// TwinCAT 3 PLC project PLC
// ProgramVersion: 3.1.4024.0
// libraries:
//   Tc2_Standard, * (Beckhoff Automation GmbH)
//   Tc2_System, * (Beckhoff Automation GmbH)
//   Tc3_Module, * (Beckhoff Automation GmbH)
// project tree:
//   / PlcTask.TcTTO
//   POUs/ MAIN.TcPOU
//   POUs/TEMPLATE ST FB%27s/ AdvancedFaultDetection.TcPOU (not stored), Auto_Manual_CycleControl.TcPOU (not stored), CYL.TcPOU (not stored), FB_analog.TcPOU (not stored), FB_Conveyor.TcPOU (not stored), FB_Fan.TcPOU (not stored), FB_FaultDetection.TcPOU (not stored), FB_FlowMeter.TcPOU (not stored), FB_IO_Card_ARRAY.TcPOU (not stored), FB_IO_CARD_BOOL.TcPOU (not stored), FB_LevelSensor.TcPOU (not stored), FB_Pump.TcPOU (not stored), FB_Sensor.TcPOU (not stored), FB_StackLight.TcPOU (not stored), FB_STATUS.TcPOU (not stored), FB_Tank.TcPOU (not stored), FB_Valve.TcPOU (not stored), FB_Valve_Proportional.TcPOU (not stored), FB_VFD_FWD_REV.TcPOU (not stored), Reject_Conveyor.TcPOU (not stored), SensorProcessing.TcPOU (not stored)
// real-time tasks:
//   TASK PlcTask: cycle T#10ms, priority 20, ADS port 350

CONFIGURATION PLC
    RESOURCE PLC ON TwinCAT3
        TASK PlcTask(INTERVAL := T#10ms, PRIORITY := 20);
        PROGRAM MAIN WITH PlcTask : MAIN;
    END_RESOURCE
END_CONFIGURATION

// ---- POUs/MAIN.TcPOU
PROGRAM MAIN
VAR
END_VAR

END_PROGRAM
